// TIA Portal V20 export
TYPE "typeCmControlNodeInterlock"
// stored: Namespace Unit1.Em10
   STRUCT
      laserMarkStageLift : "LER_typeTwoWayActuatorInterlock";
      laserMarkCover : "LER_typeTwoWayActuatorInterlock";
   END_STRUCT;
END_TYPE
